// TwinCAT 3 PLC project BasicCoR_PLC
// ProgramVersion: 3.1.4022.4
// libraries:
//   Tc2_Standard, * (Beckhoff Automation GmbH)
//   Tc2_System, * (Beckhoff Automation GmbH)
//   Tc3_Module, * (Beckhoff Automation GmbH)
// project tree:
//   Diagrams/ ClassDiagram.TcCD (not stored)
//   Handlers/FBs/ FB_BaseHandler.TcPOU, FB_StaticHandler1.TcPOU, FB_StaticHandler2.TcPOU, FB_StaticHandler3.TcPOU, FB_StaticHandler_n.TcPOU
//   Handlers/ITFs/ I_Handler.TcIO
//   / PlcTask.TcTTO
//   POUs/POUs/ MAIN.TcPOU
// real-time tasks:
//   TASK PlcTask: cycle T#10ms, priority 20, ADS port 350

CONFIGURATION BasicCoR_PLC
    RESOURCE PLC ON TwinCAT3
        TASK PlcTask(INTERVAL := T#10ms, PRIORITY := 20);
        PROGRAM MAIN WITH PlcTask : MAIN;
    END_RESOURCE
END_CONFIGURATION

// ---- Handlers/ITFs/I_Handler.TcIO
INTERFACE I_Handler

METHOD handle : BOOL
VAR_INPUT
	request	:	STRING;
END_VAR
END_METHOD

METHOD setNext : BOOL
VAR_INPUT
	h	: I_Handler;
END_VAR
END_METHOD

END_INTERFACE

// ---- POUs/POUs/MAIN.TcPOU
PROGRAM MAIN
VAR
	h1				:	FB_StaticHandler1;
	h2				:	FB_StaticHandler2;
	h3				:	FB_StaticHandler3;
	h_n				:	FB_StaticHandler_n;
	request 		:	STRING	:= 'Hello world!';
	xStartProcess	: 	BOOL;
END_VAR

h1.setNext(h2);
h2.setNext(h3);
h3.setNext(h_n);

(*************************************************************
*************SIMULATION***************************************
***
*** Leave request as "hello world!" for full chain processing
*** or use the string phrases below to interupt the chain.
***
***	Handler 1 - request := 'Handler 1 Interupt';
*** Handler 2 - request := 'Handler 2 Interupt';
*** Handler 3 - request := 'Handler 3 Interupt';
**************************************************************
*************************************************************)

IF xStartProcess THEN
	xStartProcess := FALSE;
	h1.handle(request);
END_IF

END_PROGRAM

// ---- Handlers/FBs/FB_StaticHandler1.TcPOU
FUNCTION_BLOCK FB_StaticHandler1 EXTENDS FB_BaseHandler
VAR_INPUT
END_VAR
VAR_OUTPUT
END_VAR
VAR
END_VAR

METHOD handle : BOOL
VAR_INPUT
	request	:	STRING;
END_VAR
IF request = 'Handler 1 Interupt' THEN
	ADSLOGSTR(ADSLOG_MSGTYPE_MSGBOX, request, ' ');
ELSE
	ADSLOGSTR(ADSLOG_MSGTYPE_MSGBOX, '@H1 Moving to next handler ', '');
	SUPER^.handle(request);
END_IF
END_METHOD

END_FUNCTION_BLOCK

// ---- Handlers/FBs/FB_BaseHandler.TcPOU
FUNCTION_BLOCK FB_BaseHandler IMPLEMENTS I_Handler
VAR_INPUT
END_VAR
VAR_OUTPUT
END_VAR
VAR
	next : I_Handler;
END_VAR

METHOD handle : BOOL
VAR_INPUT
	request	:	STRING;
END_VAR
IF ADR(next) <> 0 THEN
	next.handle(request);
END_IF
END_METHOD

METHOD setNext : BOOL
VAR_INPUT
	h	: I_Handler;
END_VAR
next := h;
END_METHOD

END_FUNCTION_BLOCK

// ---- Handlers/FBs/FB_StaticHandler2.TcPOU
FUNCTION_BLOCK FB_StaticHandler2 EXTENDS FB_BaseHandler
VAR_INPUT
END_VAR
VAR_OUTPUT
END_VAR
VAR
END_VAR

METHOD handle : BOOL
VAR_INPUT
	request	:	STRING;
END_VAR
IF request = 'Handler 2 Interupt' THEN
	ADSLOGSTR(ADSLOG_MSGTYPE_MSGBOX, request, ' ');
ELSE
	ADSLOGSTR(ADSLOG_MSGTYPE_MSGBOX, '@H2 Moving to next handler ', '');
	SUPER^.handle(request);
END_IF
END_METHOD

END_FUNCTION_BLOCK

// ---- Handlers/FBs/FB_StaticHandler3.TcPOU
FUNCTION_BLOCK FB_StaticHandler3 EXTENDS FB_BaseHandler
VAR_INPUT
END_VAR
VAR_OUTPUT
END_VAR
VAR
END_VAR

METHOD handle : BOOL
VAR_INPUT
	request	:	STRING;
END_VAR
IF request = 'Handler 3 Interupt' THEN
	ADSLOGSTR(ADSLOG_MSGTYPE_MSGBOX, request, ' ');
ELSE
	ADSLOGSTR(ADSLOG_MSGTYPE_MSGBOX, '@H3 Moving to next handler ', '');
	SUPER^.handle(request);
END_IF
END_METHOD

END_FUNCTION_BLOCK

// ---- Handlers/FBs/FB_StaticHandler_n.TcPOU
FUNCTION_BLOCK FB_StaticHandler_n EXTENDS FB_BaseHandler
VAR_INPUT
END_VAR
VAR_OUTPUT
END_VAR
VAR
END_VAR

METHOD handle : BOOL
VAR_INPUT
	request	:	STRING;
END_VAR
ADSLOGSTR(ADSLOG_MSGTYPE_MSGBOX, request , '');
END_METHOD

END_FUNCTION_BLOCK
